FUNCTION_BLOCK FB_DataFlowManagement
VAR CONSTANT
END_VAR
//NovRam
VAR RETAIN
	NovRamData:ST_NovRam;
END_VAR
VAR_INPUT
	eDBID		: E_DBID := E_DBID.RemoteDB;
	wsDBname	: WSTRING(128); // DB Name
	stMachineInfo : ST_MachineInformation;
	stSoInfo	: ST_ShopOrderInformation;
END_VAR
VAR_OUTPUT
END_VAR
VAR
	//{attribute 'hide'}
	lrFileUseRate: ARRAY[0..6] OF LREAL;
	//{attribute 'hide'}
	lrRamUseRate:ARRAY[0..6] OF LREAL;
	
	//Data To NovRam
	//{attribute 'hide'}
	fbDataToNovRam : FB_DataToNovRam;
	//NovRam To FileRingBuffer
	//{attribute 'hide'}
	fbNovRamToFileRingBuffer:ARRAY [0..6] OF ARRAY[0..GVL.NovRamBufferRatio-1] OF FB_NovRamToFileRingBuffer;
	//FileRingBuffer To DataBase
	//{attribute 'hide'}
	fbFileRingBufferToDB:ARRAY [0..6] OF ARRAY [0..GVL.NovRamBufferRatio-1] OF ARRAY[0..GVL.FileRingBufferRatio-1] OF FB_FileRingBufferToDB;
END_VAR

//FB cyclic
M_CyclicUpdate();

//Calc Use Rate
M_CalcUseRate(lrFileUseRate:=lrFileUseRate,lrRamUseRate:=lrRamUseRate);

METHOD M_Add_AlarmHistory : BOOL
VAR_INPUT
	addData : ST_AlarmInfo_DB ;
END_VAR
M_Add_AlarmHistory:=fbDataToNovRam.M_AlarmHistory(addData:=addData);
END_METHOD

METHOD M_Add_ProductionHistoryInspection : BOOL
VAR_INPUT
	addData:ST_PHI_GroupData_DB;
END_VAR
M_Add_ProductionHistoryInspection:=fbDataToNovRam.M_ProductionHistory(addData:=addData);
END_METHOD

METHOD M_Add_ProductionReport : BOOL
VAR_INPUT
	addData:ST_OEE_ProductionReport;
END_VAR
M_Add_ProductionReport:=fbDataToNovRam.M_ProductionReport(addData:=addData);
END_METHOD

METHOD M_Add_ProductionSummary : BOOL
VAR_INPUT
	addData:ST_OEE_ProductionSummary;
END_VAR
M_Add_ProductionSummary:=fbDataToNovRam.M_ProductionSummary(addData:=addData);
END_METHOD

METHOD M_Add_RegularCheckResults : BOOL
VAR_INPUT
	addData:ST_RegularCheck_Results;
END_VAR
M_Add_RegularCheckResults:=fbDataToNovRam.M_RegularCheckResults(addData:=addData);
END_METHOD

METHOD M_Add_SoDuration : BOOL
VAR_INPUT
	addData:ST_SoDuration;
END_VAR
M_Add_SoDuration:=fbDataToNovRam.M_SoDuration(addData:=addData);
END_METHOD

METHOD M_Add_StopCount : BOOL
VAR_INPUT
	addData:ST_StopCount;
END_VAR
M_Add_StopCount:=fbDataToNovRam.M_StopCount(addData:=addData);
END_METHOD

METHOD M_AutoFill_MachineInfo : BOOL
VAR_INPUT
	refsFaam_id		: REFERENCE TO STRING(20); // 設備ID
	refwsEquipment : REFERENCE TO WSTRING(25); // 設備名稱
END_VAR
(*
IF __ISVALIDREF(refwsEquipment) AND_THEN refwsEquipment = "" THEN //檢查Equipmet是否有填值
	refwsEquipment := stMachineInfo.wsEquipment;
END_IF

IF __ISVALIDREF(refsFaam_id) AND_THEN refsFaam_id = '' THEN //檢查Equipmet是否有填值
	refsFaam_id := stMachineInfo.sFaam_id;
END_IF

M_AutoFill_MachineInfo := True;
*)
END_METHOD

METHOD M_AutoFill_SoInfo : BOOL
VAR_INPUT
	refdiSo_id	: REFERENCE TO DINT;
	refsSo_number : REFERENCE TO STRING(12);
END_VAR
(*
IF __ISVALIDREF(refdiSo_id) AND_THEN refdiSo_id = 0 THEN
	refdiSo_id := stSoInfo.diSo_id;
END_IF

IF __ISVALIDREF(refsSo_number) AND_THEN refsSo_number = '' THEN
	refsSo_number := stSoInfo.sSo_number;
END_IF

M_AutoFill_SoInfo := True;
*)
END_METHOD

METHOD PRIVATE M_CalcUseRate : BOOL
VAR_IN_OUT
	lrFileUseRate: ARRAY[0..6] OF LREAL;
	lrRamUseRate:ARRAY[0..6] OF LREAL;
END_VAR
VAR
	iStruType:UDINT;
	iRamIndex:UDINT;iFileIndex:UDINT;
	
	udiRamFullCount:UDINT;
	udiFileFullCount:UDINT;
END_VAR
FOR iStruType:=0 TO 6 DO
	
	udiRamFullCount:=0;
	udiFileFullCount:=0;
	
	FOR iRamIndex:=0 TO GVL.NovRamBufferRatio-1 DO
		
		IF NovRamData.arrNovRam_Status[iStruType].RowDataLocked[iRamIndex] THEN//ram
			udiRamFullCount:=udiRamFullCount+1;
		END_IF
		
		FOR iFileIndex:=0 TO GVL.FileRingBufferRatio-1 DO//file
			IF NovRamData.arrFileRingBuffer_Status[iStruType].bFileFull[iRamIndex][iFileIndex] = TRUE THEN
				udiFileFullCount:=udiFileFullCount+1;
			END_IF
		END_FOR
	END_FOR
	
	lrFileUseRate[iStruType]:=UDINT_TO_LREAL(udiFileFullCount) 
								/ (UDINT_TO_LREAL(GVL.NovRamBufferRatio) * UDINT_TO_LREAL(GVL.FileRingBufferRatio));
	lrRamUseRate[iStruType]:=UDINT_TO_LREAL(udiRamFullCount) / UDINT_TO_LREAL(GVL.NovRamBufferRatio);
END_FOR
END_METHOD

METHOD PRIVATE M_CyclicUpdate : BOOL
VAR_INPUT
END_VAR
VAR
	i:UDINT;k:UDINT;
END_VAR
//Data to NovRam
fbDataToNovRam(NovRamData:=NovRamData);


//NovRam to File
FOR i:= 0 TO GVL.NovRamBufferRatio-1 DO
	fbNovRamToFileRingBuffer[E_DB_StructureType.AlarmHistory][i](udiNovRamIndex:=i,dataType:=E_DB_StructureType.AlarmHistory,NovRamData:=NovRamData);
	fbNovRamToFileRingBuffer[E_DB_StructureType.ProductionHistory][i](udiNovRamIndex:=i,dataType:=E_DB_StructureType.ProductionHistory,NovRamData:=NovRamData);
	fbNovRamToFileRingBuffer[E_DB_StructureType.ProductionReport][i](udiNovRamIndex:=i,dataType:=E_DB_StructureType.ProductionReport,NovRamData:=NovRamData);
	fbNovRamToFileRingBuffer[E_DB_StructureType.ProductionSummary][i](udiNovRamIndex:=i,dataType:=E_DB_StructureType.ProductionSummary,NovRamData:=NovRamData);
	fbNovRamToFileRingBuffer[E_DB_StructureType.SoDuration][i](udiNovRamIndex:=i,dataType:=E_DB_StructureType.SoDuration,NovRamData:=NovRamData);
	fbNovRamToFileRingBuffer[E_DB_StructureType.StopCount][i](udiNovRamIndex:=i,dataType:=E_DB_StructureType.StopCount,NovRamData:=NovRamData);
	fbNovRamToFileRingBuffer[E_DB_StructureType.RegularCheckResults][i](udiNovRamIndex:=i,dataType:=E_DB_StructureType.RegularCheckResults,NovRamData:=NovRamData);
	
END_FOR
//File to DB
FOR i:=0 TO gvl.NovRamBufferRatio-1 DO
	FOR k:=0 TO GVL.FileRingBufferRatio-1 DO
		
		fbFileRingBufferToDB[E_DB_StructureType.AlarmHistory][i][k](udiNovRam_BufferIndex:=i,udiFile_Index:=k,dataType:=E_DB_StructureType.AlarmHistory,NovRamData:=NovRamData);
		fbFileRingBufferToDB[E_DB_StructureType.ProductionHistory][i][k](udiNovRam_BufferIndex:=i,udiFile_Index:=k,dataType:=E_DB_StructureType.ProductionHistory,NovRamData:=NovRamData);
		fbFileRingBufferToDB[E_DB_StructureType.ProductionReport][i][k](udiNovRam_BufferIndex:=i,udiFile_Index:=k,dataType:=E_DB_StructureType.ProductionReport,NovRamData:=NovRamData);
		fbFileRingBufferToDB[E_DB_StructureType.ProductionSummary][i][k](udiNovRam_BufferIndex:=i,udiFile_Index:=k,dataType:=E_DB_StructureType.ProductionSummary,NovRamData:=NovRamData);
		fbFileRingBufferToDB[E_DB_StructureType.SoDuration][i][k](udiNovRam_BufferIndex:=i,udiFile_Index:=k,dataType:=E_DB_StructureType.SoDuration,NovRamData:=NovRamData);
		fbFileRingBufferToDB[E_DB_StructureType.StopCount][i][k](udiNovRam_BufferIndex:=i,udiFile_Index:=k,dataType:=E_DB_StructureType.StopCount,NovRamData:=NovRamData);
		fbFileRingBufferToDB[E_DB_StructureType.RegularCheckResults][i][k](udiNovRam_BufferIndex:=i,udiFile_Index:=k,dataType:=E_DB_StructureType.RegularCheckResults,NovRamData:=NovRamData);
		
	END_FOR
END_FOR
END_METHOD

END_FUNCTION_BLOCK

(* stored: Version 1.1.0.1, ProductVersion 3.1.4024.11
   POU FB_DataFlowManagement: Id {f7d5b7fb-9a05-4d0d-a367-7c2a7531c7d8}, SpecialFunc None
   Folder Add: Id {cf7edd92-eecd-48da-b39e-1de52b16613d}
   Folder Sub: Id {54692b75-075a-41bc-bde4-34a4d1eaeeff}
   Folder Private: Id {15d896e7-5dd7-4dee-a796-c8fa327031aa}
   Method M_Add_AlarmHistory: Id {ab3fc6a2-e2f0-4d96-9438-03f3cf2e8e90}
   Method M_Add_ProductionHistoryInspection: Id {5e6c14bf-c6c2-43f8-923f-2e95c0af200a}
   Method M_Add_ProductionReport: Id {ff1625e1-b646-4af9-ad66-f6b62dc7a7e1}
   Method M_Add_ProductionSummary: Id {3838ca8f-0ad7-46eb-9f0e-7d065e2f16dd}
   Method M_Add_RegularCheckResults: Id {2944582c-7086-467c-9f74-6b78da24712f}
   Method M_Add_SoDuration: Id {5d8d8a5e-7fd4-4d7e-823f-3bad764c7d9d}
   Method M_Add_StopCount: Id {d7560351-6982-4cf3-817b-5f091a468833}
   Method M_AutoFill_MachineInfo: Id {f4898d49-910f-400a-bf4f-5f42df858981}
   Method M_AutoFill_SoInfo: Id {3f245a41-a756-4e39-a2ca-b846a05ac8e0}
   Method M_CalcUseRate: Id {b1b25544-751d-4a1e-a1ef-1e90150db345}
   Method M_CyclicUpdate: Id {e14d3aed-0555-49d4-9fa9-9256ac3db4b1} *)
